(* PLC project Untitled47, Machine Expert Logic Builder V21.0.22.0, author SESA640032 *)
(* stored: creationDateTime 2023-06-02T14:15:08.4823286, version 0.0.0.0, modificationDateTime 2023-06-02T10:41:04.8480725 *)

PROGRAM SR_TcpClient
  VAR
    sIpAddrServer : STRING(15);  (* IP address of the TCP server *)
    uiTcpServerPort : UINT;  (* Port of the TCP server *)
    stTlsSettings : TcpUdp.ST_TlsSettingsClient;
    xUseTls : BOOL;
    xComInProgress : BOOL;  (* indicates the TCP communication is in progress *)
    etTcpClientState : TCPUDP.ET_State;  (* state of the TCP connection *)
    etTcpClientResult : TCPUDP.ET_Result;  (* result of the latest method call *)
    xInterruptEth : BOOL;  (* indicates the Ethernet was disturbed, while the TCP com. was in progress *)
    xConnectDone : BOOL;  (* flag indicates the result of the method Connect *)
    xCloseDone : BOOL;  (* flag indicates the result of the method Close *)
    udiSentData : UDINT;  (* Number of bytes sent to the server using the method Send *)
    udiPeekedData : UDINT;  (* Number of bytes peeked from the buffre using the method Peek *)
    udiSizeReceivedData : UDINT;  (* Number of bytes read from the buffer using the method Receive *)
    xAlarmConnect : BOOL;  (* Alarm: connection failed *)
    xAlarmSend : BOOL;  (* Alarm: not all bytes have been sent *)
    xAlarmPeek : BOOL;  (* Alarm: Peek method *)
    xAlarmReceive : BOOL;  (* Alarm: Receive method *)
    xAlarmTimeout : BOOL;  (* Alarm: Timeout waiting for response *)
    xAlarmClose : BOOL;  (* Alarm: Close method *)
    xWarnLenOfDataReceived : BOOL;  (* Warning: Data length in received data doesn't meet the number of bytes available to read *)
    xWarnPeerDisconnect : BOOL;  (* Warning: Peer has disconnected *)
    xDiag : BOOL;  (* Indicates a Diag message is available *)
    sDiagMessage : STRING;  (* Diag message created from the alarms and warnings *)
    sStepFailed : STRING;  (* String contains the name of the Step or Method which is failed to precise the result message *)
    xDataOkay : BOOL;  (* Check of transmission ID okay, received data are valid *)
    stDataSend : ST_Data;
    stDataReceive : ST_Data;
    abySendBuffer : ARRAY[0..(SIZEOF(stDataSend) - 1)] OF BYTE;  (* send buffer *)
    abyReceiveBuffer : ARRAY[0..(SIZEOF(stDataReceive) - 1)] OF BYTE;  (* receive buffer *)
    iState : INT;  (* current state of the staemachine *)
    udiFillLevelSend : UDINT;  (* fill level of the send buffer *)
    uiCountSendings : UINT;
    udiFillLevelReceive : UDINT;  (* fill level of the receive buffer *)
    udiReceiveBufferSize : UDINT;  (* max number of Bytes to be read using the Receive method, !!! Must not greater than the Buffer size! !!! *)
    timTimeoutReceive : TIME := TIME#10s0ms;  (* time to wait for the response from the server before closing the connection with timeout alarm *)
    timStartWaiting : TIME;  (* reference time for timeout monitoring *)
    fbTcpClient : TCPUDP.FB_TCPClient2;  (* FB Instance *)
    fbRTrigStart : Standard.R_TRIG;
    fbRTrigClearResult : Standard.R_TRIG;
    timLastComCycle : TIME;  (* duration of last successful communication cycle *)
    timStartCom : TIME;  (* reference time for communication cycle measurement *)
    xFirstCycle : BOOL := TRUE;  (* indicates the first cycle of the program after a warmstart *)
  END_VAR

            (* Check the Ethernet Status of the controller *)
IF NOT GVL.g_xEthReady THEN
	xInterruptEth	:= xComInProgress;
	xComInProgress	:= FALSE;	// reset the status flag
	iState			:= 100;	// go into state 100 - do nothing
ELSE
	IF (iState = 100) THEN
		IF (fbTcpClient.State <> TCPUDP.ET_State.Idle) THEN
			iState	:= 50;
		ELSE
			iState	:= 0;
		END_IF
	END_IF
	xInterruptEth	:= FALSE;
END_IF 

(* Visu variables - inputs *)
// Monitor rising edges of commands *)
fbRTrigStart		(CLK:= GVL_VisuTcpClient.g_xCmdStart);
fbRTrigClearResult	(CLK:= GVL_VisuTcpClient.g_xCmdClearResult);
IF (iState = 0) OR xFirstCycle THEN
	// only in state "wait for command" the input from the visu is accepted
	stDataSend.sData	:= GVL_VisuTcpClient.g_stDataToSend.sData;
	timTimeoutReceive	:= GVL_VisuTcpClient.g_timTimeoutReceive;
	sIpAddrServer		:= GVL_VisuTcpClient.g_sIpAddrServer;
	uiTcpServerPort		:= GVL_VisuTcpClient.g_uiTcpServerPort;
	xUseTls							:= GVL_VisuTcpClient.g_xTlsSelected;
	stTlsSettings.etCertVerifyMode	:= GVL_VisuTcpClient.g_etCertVerifyMode;
ELSE
	// update the visu input while communication is in progress
	GVL_VisuTcpClient.g_stDataToSend.sData	:= stDataSend.sData;
	GVL_VisuTcpClient.g_timTimeoutReceive	:= timTimeoutReceive;
	GVL_VisuTcpClient.g_sIpAddrServer		:= sIpAddrServer;
	GVL_VisuTcpClient.g_uiTcpServerPort		:= uiTcpServerPort;
END_IF

(* Clear the result *)
IF (fbRTrigClearResult.Q OR (fbRTrigStart.Q AND iState = 0)) THEN
	// reset all alarms and warnings
	xAlarmConnect			:= FALSE;
	xAlarmSend				:= FALSE;
	xAlarmPeek				:= FALSE;
	xAlarmReceive			:= FALSE;
	xAlarmTimeout			:= FALSE;
	xAlarmClose				:= FALSE;
	xWarnLenOfDataReceived	:= FALSE;
	xWarnPeerDisconnect		:= FALSE;
	
	fbTcpClient.ResetResult();
	etTcpClientResult		:= TCPUDP.ET_Result.Ok;
	sStepFailed				:='';
END_IF

(* TCP Client state *)
etTcpClientState		:= fbTcpClient.State;

(* State machine *)
CASE iState OF
	0: (* Wait for command to connect *)
		IF xComInProgress THEN
			xComInProgress	:= FALSE;
			timLastComCycle	:= SEL(xDiag,(TIME()- timStartCom),timLastComCycle);
		END_IF
		
		IF (etTcpClientState <> TCPUDP.ET_State.Idle) THEN
			iState	:= 50;	// not ready for connect, first perform a Close command
			
		ELSIF fbRTrigStart.Q THEN
			(* init variables *)
			uiCountSendings		:= 0;
			timStartCom			:= TIME();
			// init the receive buffer
			SysMem.SysMemSet(pDest:=ADR(abyReceiveBuffer),udiValue:=0,udiCount:=SIZEOF(abyReceiveBuffer));
			SysMem.SysMemSet(pDest:=ADR(stDataReceive),udiValue:=0,udiCount:=SIZEOF(stDataReceive));
			
			(* Connect to server *)
			IF NOT xUseTls THEN
				xConnectDone	:= fbTcpClient.Connect(	i_sServerIP		:= sIpAddrServer,
														i_uiServerPort	:= uiTcpServerPort);
			ELSE
				xConnectDone	:= fbTcpClient.ConnectTls(	i_sServerIP		:= sIpAddrServer,
															i_uiServerPort	:= uiTcpServerPort,
															i_stTlsSettings := stTlsSettings);
			END_IF			

	
			IF xConnectDone THEN
				iState				:= 10;	// wait for the connection
				xComInProgress		:= TRUE;
			ELSE
				etTcpClientResult	:= fbTcpClient.Result;	// connection failed, check the result
				sStepFailed			:= 'Connect: ';
				xAlarmConnect		:= TRUE;
			END_IF
			
		END_IF		
	
	10:	(* Connection in progress *)
		IF (etTcpClientState <> TCPUDP.ET_State.Connecting) THEN
			IF (etTcpClientState = TCPUDP.ET_State.Connected) THEN
				iState	:= 20;	// TCP server is connected
			ELSE
				etTcpClientResult	:= fbTcpClient.Result;	// connection failed, check the result
				sStepFailed			:= 'Connect: ';
				xAlarmConnect		:= TRUE;
				iState				:= 50;					// connection failed, close the socket
			END_IF
		END_IF
	
	20:	(* TCP Server is connected -> Send data *)
		A20_Send();
	
	30:	(* Response from TCP server is expected *)
		A30_Receive();
				
	//40:	(* Shutdown - no more data will be sent *)
	//	shutdown not implemented
			
	50:	(* Close the connection/socket due to an error during Connect *)
		xCloseDone	:= fbTcpClient.Close();
		iState	:= 0;	// go to wait for command
		
	100:(* Ethernet Interface of the controller not ready *)
		;	// do nothing
		
END_CASE

(* Create diagnostic message *)
IF (iState = 100) THEN		
	sDiagMessage	:= 'Ethernet link not ready';
	xDiag			:= TRUE;	
ELSIF xAlarmConnect THEN		
	sDiagMessage	:= 'Connection failed';
	xDiag			:= TRUE;
ELSIF xAlarmSend THEN		
	sDiagMessage	:= 'Send data failed';
	xDiag			:= TRUE;
ELSIF xAlarmPeek THEN		
	sDiagMessage	:= 'Peeking received data failed';
	xDiag			:= TRUE;
ELSIF xAlarmReceive THEN		
	sDiagMessage	:= 'No data could be read';
	xDiag			:= TRUE;
ELSIF xAlarmTimeout THEN		
	sDiagMessage	:= 'Timeout while waiting for response';
	xDiag			:= TRUE;
ELSIF xAlarmClose THEN		
	sDiagMessage	:= 'Close connection failed';
	xDiag			:= TRUE;
ELSIF xWarnLenOfDataReceived THEN		
	sDiagMessage	:= 'Length of received data inconsistant';
	xDiag			:= TRUE;
ELSIF xWarnPeerDisconnect THEN		
	sDiagMessage	:= 'Peer has disconnected';
	xDiag			:= TRUE;
ELSE			
	sDiagMessage	:= 'No alarm or warning';
	xDiag			:= FALSE;
END_IF

(* Visu variables - outputs *)
GVL_VisuTcpClient.g_sTcpClientState				:= TCPUDP.FC_EtStateToString(i_etState:= etTcpClientState);
GVL_VisuTcpClient.g_sTcpClientResult			:= Standard.CONCAT(sStepFailed, TCPUDP.FC_EtResultToString(i_etResult:= etTcpClientResult));
GVL_VisuTcpClient.g_stDataToSend.uiTransId		:= stDataSend.uiTransId;
GVL_VisuTcpClient.g_stDataToSend.usiLenOfData	:= stDataSend.usiLenOfData;
GVL_VisuTcpClient.g_stDataReceived.uiTransId	:= stDataReceive.uiTransId;
GVL_VisuTcpClient.g_stDataReceived.usiLenOfData	:= stDataReceive.usiLenOfData;
GVL_VisuTcpClient.g_stDataReceived.sData		:= stDataReceive.sData;
GVL_VisuTcpClient.g_xComInProgress				:= xComInProgress;
GVL_VisuTcpClient.g_xDiag						:= xDiag;
GVL_VisuTcpClient.g_sDiagMessage				:= sDiagMessage;
GVL_VisuTcpClient.g_timLastComCycle				:= timLastComCycle;
GVL_VisuTcpClient.g_xTlsSelected				:= xUseTls;
GVL_VisuTcpClient.g_sCertVerifyMode				:= TCPUDP.FC_EtCertVerifyModeToString(stTlsSettings.etCertVerifyMode);

(* reset the first cycle information *)
xFirstCycle	R= xFirstCycle;
          

ACTION A30_Receive:
                (* Response from TCP server is expected *)	
IF fbTcpClient.PeerHasDisconnected THEN
	// Peer has diconnected
	xWarnPeerDisconnect	:= TRUE;
	iState				:= 50;	// close the connection
	
ELSIF fbTcpClient.IsReadable THEN
	xDataOkay	:= FALSE;	// reset the flag
	// take a peek on the received data
	udiPeekedData	:= fbTcpClient.Peek(i_pbyReceiveBuffer		:= ADR(abyReceiveBuffer),
										i_udiReceiveBufferSize	:= 3);
	// check the result of peek			
	IF (udiPeekedData = 3) THEN
		stDataReceive.uiTransId		:= abyReceiveBuffer[0];
		stDataReceive.uiTransId		:= SHL(stDataReceive.uiTransId,8) OR abyReceiveBuffer[1];
		stDataReceive.usiLenOfData	:= abyReceiveBuffer[2];
		xDataOkay					:= (stDataSend.uiTransId = stDataReceive.uiTransId);
	ELSE
		etTcpClientResult	:= fbTcpClient.Result;	// Peek failed, check the result
		sStepFailed			:= 'Peek: ';
		xAlarmPeek			:= TRUE;
	END_IF
	
	IF xDataOkay THEN
		// set the data to be read from the buffer, NOTE: 2048 bytes is the limitation for M241 & M251 controllers
		udiReceiveBufferSize	:= LIMIT(1, MIN(SIZEOF(abyReceiveBuffer), (stDataReceive.usiLenOfData + 3)), 2048);
		
		// take the data from the buffer using the Receive method
		udiFillLevelReceive	:=	0;	// initialize the fill-level
		udiSizeReceivedData	:= fbTcpClient.Receive(	i_pbyReceiveBuffer		:= ADR(abyReceiveBuffer),
													i_udiReceiveBufferSize	:= udiReceiveBufferSize,
													iq_udiFillLevel			:= udiFillLevelReceive);
		
		IF (udiSizeReceivedData = 0) OR (fbTcpClient.Result <> TCPUDP.ET_Result.Ok) THEN
			etTcpClientResult	:= fbTcpClient.Result;	// Peek failed, check the result
			sStepFailed			:= 'Receive: ';
			xAlarmReceive		:= TRUE;
		ELSE
		// convert the data to string
		TCPUDP.FC_ReadSTRING(	i_pbyBuffer		:= ADR(abyReceiveBuffer[3]),
								i_psString		:= ADR(stDataReceive.sData),
								i_uiMaxLength	:= SIZEOF(stDataReceive.sData)-1,
								i_xStopAtZero	:= TRUE);
			
		END_IF
	ELSE
		// Unknown data
		stDataReceive.sData	:= 'Invalid TransmissionID';
	END_IF
	iState				:= 50;	// close the connection
					
ELSIF ((TIME() - timStartWaiting) > timTimeoutReceive) THEN
	// Timeout while waiting for response
	xAlarmTimeout	:= TRUE;
	iState			:= 50;	// close the connection
END_IF
              
END_ACTION

ACTION A20_Send:
                (* TCP Server is connected -> Send data *)
IF (udiFillLevelSend = 0) THEN
	// prepare data to send: Transmission ID (2 Bytes), Length of Data (1 byte), and Data (STRING)
	stDataSend.uiTransId	:=TIME_TO_UINT(TIME());
	stDataSend.usiLenOfData	:=INT_TO_BYTE(Standard.LEN(stDataSend.sData)+1);
	
	abySendBuffer[0] :=UINT_TO_BYTE(SHR(stDataSend.uiTransId,8));
	abySendBuffer[1] :=UINT_TO_BYTE(stDataSend.uiTransId);
	abySendBuffer[2] :=stDataSend.usiLenOfData;
	TCPUDP.FC_WriteSTRING(	i_pbyBuffer		:= ADR(abySendBuffer[3]),
							i_psString		:= ADR(stDataSend.sData),
							i_uiMaxLength	:= SIZEOF(abySendBuffer)-3);
							
	// determine the number of bytes to be sent, NOTE: 2048 bytes is the limitation for M241 & M251 controllers
	udiFillLevelSend := MIN((stDataSend.usiLenOfData + 3), 2048);
END_IF

// send data
udiSentData	:= fbTcpClient.Send(i_pbySendBuffer	:= ADR(abySendBuffer),
								iq_udiFillLevel	:= udiFillLevelSend);
					
// count the number of Send calls
uiCountSendings	:= uiCountSendings + 1;
		
// check the result of sending
IF (udiSentData = 0) OR (fbTcpClient.Result <> TCPUDP.ET_Result.Ok) THEN	
	// no data have been sent
	etTcpClientResult	:= fbTcpClient.Result;	// transmission failed, check the result
	sStepFailed			:= 'Send: ';
	xAlarmSend			:= TRUE;	// set an alarm
	iState				:= 50;		// go to close
ELSIF (udiFillLevelSend > 0) THEN
	// not all data have been sent, remaining data will be sent in the next scan
	;
ELSIF (udiFillLevelSend = 0) THEN
	// all data have been sent
	iState			:= 30;		// all data have been sent, go to receive
	timStartWaiting	:= TIME();	// initialize the timer
END_IF

IF (iState <> 20) THEN
	// when leaving this state initialize the variables
	udiFillLevelSend	:= 0;
END_IF
              
END_ACTION
END_PROGRAM
